# EPICS autosave request: coaxLinkApp/Db/coaxLink_settings.req
$(P)$(R)ArrayCallbacks
$(P)$(R)DataType
$(P)$(R)SensorBitDepth
$(P)$(R)Width+R
$(P)$(R)Height+R
$(P)$(R)CameraControlMethod
$(P)$(R)SizeX
$(P)$(R)SizeY
